// Mitsubishi GX Works2 project: PULSE_EX1   PLC: Q03UDV

PROGRAM MAIN
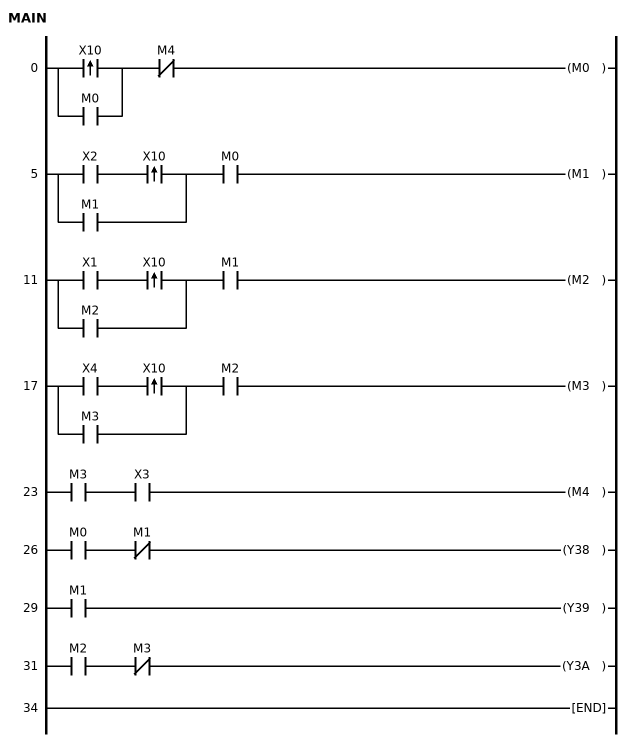
0     LDP     X10
      OR      M0
      ANI     M4
      OUT     M0
5     LD      X2
      ANDP    X10
      OR      M1
      AND     M0
      OUT     M1
11    LD      X1
      ANDP    X10
      OR      M2
      AND     M1
      OUT     M2
17    LD      X4
      ANDP    X10
      OR      M3
      AND     M2
      OUT     M3
23    LD      M3
      AND     X3
      OUT     M4
26    LD      M0
      ANI     M1
      OUT     Y38
29    LD      M1
      OUT     Y39
31    LD      M2
      ANI     M3
      OUT     Y3A
34    END
END_PROGRAM
